(* PLC project {{LIBRARY}}.{{NAME}} Demo, tc3-libraries-kb TwinCAT 3.1 *)
(* stored: creationDateTime {{TIMESTAMP}}, modificationDateTime {{TIMESTAMP}} *)

PROGRAM P_Demo_{{NAME}}
  VAR
    fb{{NAME}} : {{NAME}};
  END_VAR

            // ============================================================
// {{LIBRARY}}.{{NAME}} 演示程序
// ============================================================
// 验证步骤：
//   1. 把本 PROGRAM 加到 PlcTask 调用列表
//   2. 编译并登录目标
//   3. 在线监视 ...（输出变量）
//   4. ...（具体测试操作）
// ============================================================

{{ST_CODE}}

          
END_PROGRAM
